// TIA Portal V17 export
// export: Created 2023-05-12T10:40:25.6107869Z, DisplayName Totally Integrated Automation Portal, DisplayVersion V17 Update 4, DisplayName TIA Portal Openness, DisplayVersion V17 Update 4, DisplayName TIA Portal Version Control Interface, DisplayVersion V17, DisplayName STEP 7 Professional, DisplayVersion V17 Update 4, DisplayName STEP 7 Safety, DisplayVersion V17, DisplayName WinCC Advanced / Unified PC, DisplayVersion V17 Update 4
FUNCTION_BLOCK "FB_EM_InputConditioning"   // FB19, LAD
{ S7_Optimized_Access := 'TRUE' }
VERSION : 0.1
// stored: AutoNumber true, CodeModifiedDate 2023-05-12T12:59:41.6492354Z, CompileDate 2023-05-12T12:59:41.6492354Z, CreationDate 2023-05-08T12:19:11.3376827Z, DownloadWithoutReinit false, HandleErrorsWithinBlock false, InterfaceModifiedDate 2023-05-12T12:59:19.7337351Z, IsConsistent true, IsIECCheckEnabled false, IsKnowHowProtected false, IsRetainMemResEnabled false, IsWriteProtected false, LibraryConformanceStatus Warning: The object contains access to global data blocks., MemoryReserve 100, ModifiedDate 2023-05-12T12:59:41.6492354Z, ParameterModified 2022-09-13T10:25:33.4387708Z, PLCSimAdvancedSupport true, SetENOAutomatically false, StructureModified 2023-05-12T12:59:19.7337351Z, UDAEnableTagReadback false
   VAR
      TT01_TempZasil_PLD3_Inst { S7_SetPoint := 'True'} : "FB_CM_MeasurementPoint";
      TT02_TempPowr_PLD3_Inst { S7_SetPoint := 'True'} : "FB_CM_MeasurementPoint";
      PT01_CisnZasil_PLD3_Inst { S7_SetPoint := 'True'} : "FB_CM_MeasurementPoint";
      PT02_CisnPowr_PLD3_Inst { S7_SetPoint := 'True'} : "FB_CM_MeasurementPoint";
      PT03_CisnZasil_JKK20_Inst { S7_SetPoint := 'True'} : "FB_CM_MeasurementPoint";
      PT04_CisnPowr_JKK20_Inst { S7_SetPoint := 'True'} : "FB_CM_MeasurementPoint";
      TTs_TempSzafy_Inst { S7_SetPoint := 'True'} : "FB_CM_MeasurementPoint";
      TTk_TempKom_Inst { S7_SetPoint := 'True'} : "FB_CM_MeasurementPoint";
      TTz_TempZewn_Inst { S7_SetPoint := 'True'} : "FB_CM_MeasurementPoint";
      Rezerwa1_Inst { S7_SetPoint := 'True'} : "FB_CM_MeasurementPoint";
      Rezerwa2_Inst { S7_SetPoint := 'True'} : "FB_CM_MeasurementPoint";
      Rezerwa3_Inst { S7_SetPoint := 'True'} : "FB_CM_MeasurementPoint";
   END_VAR
BEGIN

REGION Network 1: TT01_TempZasil_PLD3 - Temperatura zasilania z PLD3
   // TT01_TempZasil_PLD3 - Temperatura zasilania z PLD3
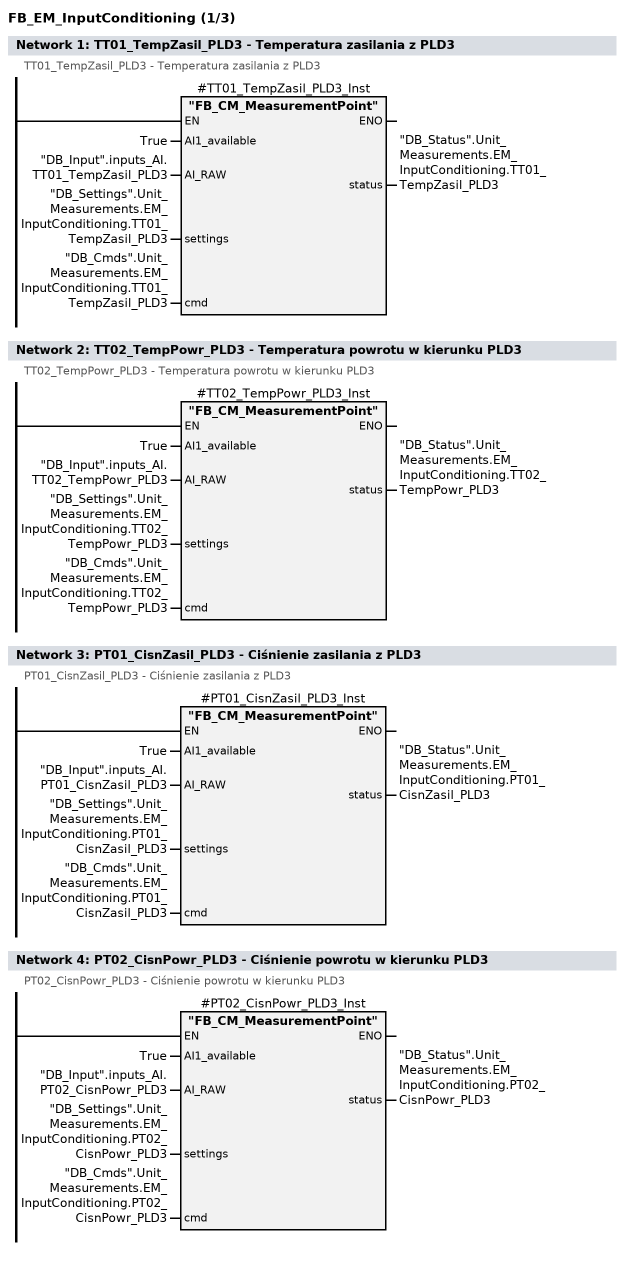
   RUNG wire#powerrail
      #TT01_TempZasil_PLD3_Inst(AI1_available := True, AI_RAW := "DB_Input".inputs_AI.TT01_TempZasil_PLD3, settings := "DB_Settings".Unit_Measurements.EM_InputConditioning.TT01_TempZasil_PLD3, cmd := "DB_Cmds".Unit_Measurements.EM_InputConditioning.TT01_TempZasil_PLD3, status => "DB_Status".Unit_Measurements.EM_InputConditioning.TT01_TempZasil_PLD3)
   END_RUNG
   // the same network as SCL:
   #TT01_TempZasil_PLD3_Inst(AI1_available := True,   // "FB_CM_MeasurementPoint"
                           AI_RAW := "DB_Input".inputs_AI.TT01_TempZasil_PLD3,
                           settings := "DB_Settings".Unit_Measurements.EM_InputConditioning.TT01_TempZasil_PLD3,
                           cmd := "DB_Cmds".Unit_Measurements.EM_InputConditioning.TT01_TempZasil_PLD3,
                           status => "DB_Status".Unit_Measurements.EM_InputConditioning.TT01_TempZasil_PLD3);
END_REGION

REGION Network 2: TT02_TempPowr_PLD3 - Temperatura powrotu w kierunku PLD3
   // TT02_TempPowr_PLD3 - Temperatura powrotu w kierunku PLD3
   RUNG wire#powerrail
      #TT02_TempPowr_PLD3_Inst(AI1_available := True, AI_RAW := "DB_Input".inputs_AI.TT02_TempPowr_PLD3, settings := "DB_Settings".Unit_Measurements.EM_InputConditioning.TT02_TempPowr_PLD3, cmd := "DB_Cmds".Unit_Measurements.EM_InputConditioning.TT02_TempPowr_PLD3, status => "DB_Status".Unit_Measurements.EM_InputConditioning.TT02_TempPowr_PLD3)
   END_RUNG
   // the same network as SCL:
   #TT02_TempPowr_PLD3_Inst(AI1_available := True,   // "FB_CM_MeasurementPoint"
                           AI_RAW := "DB_Input".inputs_AI.TT02_TempPowr_PLD3,
                           settings := "DB_Settings".Unit_Measurements.EM_InputConditioning.TT02_TempPowr_PLD3,
                           cmd := "DB_Cmds".Unit_Measurements.EM_InputConditioning.TT02_TempPowr_PLD3,
                           status => "DB_Status".Unit_Measurements.EM_InputConditioning.TT02_TempPowr_PLD3);
END_REGION

REGION Network 3: PT01_CisnZasil_PLD3 - Ciśnienie zasilania z PLD3
   // PT01_CisnZasil_PLD3 - Ciśnienie zasilania z PLD3
   RUNG wire#powerrail
      #PT01_CisnZasil_PLD3_Inst(AI1_available := True, AI_RAW := "DB_Input".inputs_AI.PT01_CisnZasil_PLD3, settings := "DB_Settings".Unit_Measurements.EM_InputConditioning.PT01_CisnZasil_PLD3, cmd := "DB_Cmds".Unit_Measurements.EM_InputConditioning.PT01_CisnZasil_PLD3, status => "DB_Status".Unit_Measurements.EM_InputConditioning.PT01_CisnZasil_PLD3)
   END_RUNG
   // the same network as SCL:
   #PT01_CisnZasil_PLD3_Inst(AI1_available := True,   // "FB_CM_MeasurementPoint"
                           AI_RAW := "DB_Input".inputs_AI.PT01_CisnZasil_PLD3,
                           settings := "DB_Settings".Unit_Measurements.EM_InputConditioning.PT01_CisnZasil_PLD3,
                           cmd := "DB_Cmds".Unit_Measurements.EM_InputConditioning.PT01_CisnZasil_PLD3,
                           status => "DB_Status".Unit_Measurements.EM_InputConditioning.PT01_CisnZasil_PLD3);
END_REGION

REGION Network 4: PT02_CisnPowr_PLD3 - Ciśnienie powrotu w kierunku PLD3
   // PT02_CisnPowr_PLD3 - Ciśnienie powrotu w kierunku PLD3
   RUNG wire#powerrail
      #PT02_CisnPowr_PLD3_Inst(AI1_available := True, AI_RAW := "DB_Input".inputs_AI.PT02_CisnPowr_PLD3, settings := "DB_Settings".Unit_Measurements.EM_InputConditioning.PT02_CisnPowr_PLD3, cmd := "DB_Cmds".Unit_Measurements.EM_InputConditioning.PT02_CisnPowr_PLD3, status => "DB_Status".Unit_Measurements.EM_InputConditioning.PT02_CisnPowr_PLD3)
   END_RUNG
   // the same network as SCL:
   #PT02_CisnPowr_PLD3_Inst(AI1_available := True,   // "FB_CM_MeasurementPoint"
                           AI_RAW := "DB_Input".inputs_AI.PT02_CisnPowr_PLD3,
                           settings := "DB_Settings".Unit_Measurements.EM_InputConditioning.PT02_CisnPowr_PLD3,
                           cmd := "DB_Cmds".Unit_Measurements.EM_InputConditioning.PT02_CisnPowr_PLD3,
                           status => "DB_Status".Unit_Measurements.EM_InputConditioning.PT02_CisnPowr_PLD3);
END_REGION

REGION Network 5: PT03_CisnZasil_JKK20 - Ciśnienie zasilania w kierunku JKK20
   // PT03_CisnZasil_JKK20 - Ciśnienie zasilania w kierunku JKK20
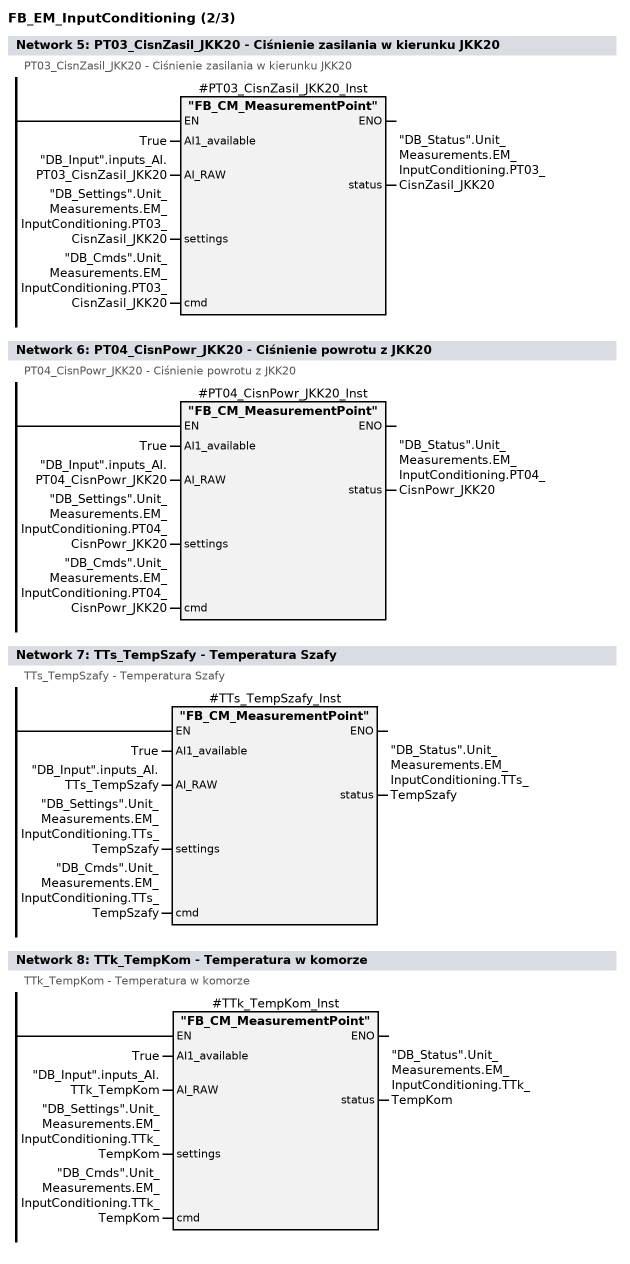
   RUNG wire#powerrail
      #PT03_CisnZasil_JKK20_Inst(AI1_available := True, AI_RAW := "DB_Input".inputs_AI.PT03_CisnZasil_JKK20, settings := "DB_Settings".Unit_Measurements.EM_InputConditioning.PT03_CisnZasil_JKK20, cmd := "DB_Cmds".Unit_Measurements.EM_InputConditioning.PT03_CisnZasil_JKK20, status => "DB_Status".Unit_Measurements.EM_InputConditioning.PT03_CisnZasil_JKK20)
   END_RUNG
   // the same network as SCL:
   #PT03_CisnZasil_JKK20_Inst(AI1_available := True,   // "FB_CM_MeasurementPoint"
                           AI_RAW := "DB_Input".inputs_AI.PT03_CisnZasil_JKK20,
                           settings := "DB_Settings".Unit_Measurements.EM_InputConditioning.PT03_CisnZasil_JKK20,
                           cmd := "DB_Cmds".Unit_Measurements.EM_InputConditioning.PT03_CisnZasil_JKK20,
                           status => "DB_Status".Unit_Measurements.EM_InputConditioning.PT03_CisnZasil_JKK20);
END_REGION

REGION Network 6: PT04_CisnPowr_JKK20 - Ciśnienie powrotu z JKK20
   // PT04_CisnPowr_JKK20 - Ciśnienie powrotu z JKK20
   RUNG wire#powerrail
      #PT04_CisnPowr_JKK20_Inst(AI1_available := True, AI_RAW := "DB_Input".inputs_AI.PT04_CisnPowr_JKK20, settings := "DB_Settings".Unit_Measurements.EM_InputConditioning.PT04_CisnPowr_JKK20, cmd := "DB_Cmds".Unit_Measurements.EM_InputConditioning.PT04_CisnPowr_JKK20, status => "DB_Status".Unit_Measurements.EM_InputConditioning.PT04_CisnPowr_JKK20)
   END_RUNG
   // the same network as SCL:
   #PT04_CisnPowr_JKK20_Inst(AI1_available := True,   // "FB_CM_MeasurementPoint"
                           AI_RAW := "DB_Input".inputs_AI.PT04_CisnPowr_JKK20,
                           settings := "DB_Settings".Unit_Measurements.EM_InputConditioning.PT04_CisnPowr_JKK20,
                           cmd := "DB_Cmds".Unit_Measurements.EM_InputConditioning.PT04_CisnPowr_JKK20,
                           status => "DB_Status".Unit_Measurements.EM_InputConditioning.PT04_CisnPowr_JKK20);
END_REGION

REGION Network 7: TTs_TempSzafy - Temperatura Szafy
   // TTs_TempSzafy - Temperatura Szafy
   RUNG wire#powerrail
      #TTs_TempSzafy_Inst(AI1_available := True, AI_RAW := "DB_Input".inputs_AI.TTs_TempSzafy, settings := "DB_Settings".Unit_Measurements.EM_InputConditioning.TTs_TempSzafy, cmd := "DB_Cmds".Unit_Measurements.EM_InputConditioning.TTs_TempSzafy, status => "DB_Status".Unit_Measurements.EM_InputConditioning.TTs_TempSzafy)
   END_RUNG
   // the same network as SCL:
   #TTs_TempSzafy_Inst(AI1_available := True,   // "FB_CM_MeasurementPoint"
                       AI_RAW := "DB_Input".inputs_AI.TTs_TempSzafy,
                       settings := "DB_Settings".Unit_Measurements.EM_InputConditioning.TTs_TempSzafy,
                       cmd := "DB_Cmds".Unit_Measurements.EM_InputConditioning.TTs_TempSzafy,
                       status => "DB_Status".Unit_Measurements.EM_InputConditioning.TTs_TempSzafy);
END_REGION

REGION Network 8: TTk_TempKom - Temperatura w komorze
   // TTk_TempKom - Temperatura w komorze
   RUNG wire#powerrail
      #TTk_TempKom_Inst(AI1_available := True, AI_RAW := "DB_Input".inputs_AI.TTk_TempKom, settings := "DB_Settings".Unit_Measurements.EM_InputConditioning.TTk_TempKom, cmd := "DB_Cmds".Unit_Measurements.EM_InputConditioning.TTk_TempKom, status => "DB_Status".Unit_Measurements.EM_InputConditioning.TTk_TempKom)
   END_RUNG
   // the same network as SCL:
   #TTk_TempKom_Inst(AI1_available := True,   // "FB_CM_MeasurementPoint"
                     AI_RAW := "DB_Input".inputs_AI.TTk_TempKom,
                     settings := "DB_Settings".Unit_Measurements.EM_InputConditioning.TTk_TempKom,
                     cmd := "DB_Cmds".Unit_Measurements.EM_InputConditioning.TTk_TempKom,
                     status => "DB_Status".Unit_Measurements.EM_InputConditioning.TTk_TempKom);
END_REGION

REGION Network 9: TTz_TempZewn - Temperatura zewnętrzna
   // TTz_TempZewn - Temperatura zewnętrzna
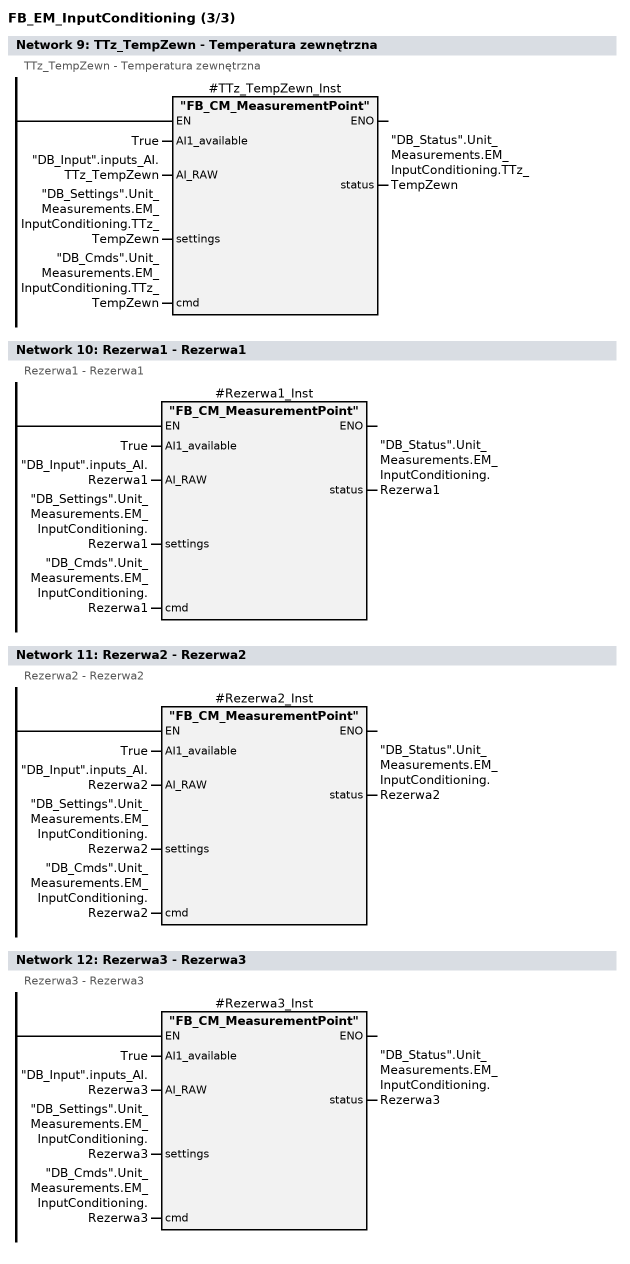
   RUNG wire#powerrail
      #TTz_TempZewn_Inst(AI1_available := True, AI_RAW := "DB_Input".inputs_AI.TTz_TempZewn, settings := "DB_Settings".Unit_Measurements.EM_InputConditioning.TTz_TempZewn, cmd := "DB_Cmds".Unit_Measurements.EM_InputConditioning.TTz_TempZewn, status => "DB_Status".Unit_Measurements.EM_InputConditioning.TTz_TempZewn)
   END_RUNG
   // the same network as SCL:
   #TTz_TempZewn_Inst(AI1_available := True,   // "FB_CM_MeasurementPoint"
                      AI_RAW := "DB_Input".inputs_AI.TTz_TempZewn,
                      settings := "DB_Settings".Unit_Measurements.EM_InputConditioning.TTz_TempZewn,
                      cmd := "DB_Cmds".Unit_Measurements.EM_InputConditioning.TTz_TempZewn,
                      status => "DB_Status".Unit_Measurements.EM_InputConditioning.TTz_TempZewn);
END_REGION

REGION Network 10: Rezerwa1 - Rezerwa1
   // Rezerwa1 - Rezerwa1
   RUNG wire#powerrail
      #Rezerwa1_Inst(AI1_available := True, AI_RAW := "DB_Input".inputs_AI.Rezerwa1, settings := "DB_Settings".Unit_Measurements.EM_InputConditioning.Rezerwa1, cmd := "DB_Cmds".Unit_Measurements.EM_InputConditioning.Rezerwa1, status => "DB_Status".Unit_Measurements.EM_InputConditioning.Rezerwa1)
   END_RUNG
   // the same network as SCL:
   #Rezerwa1_Inst(AI1_available := True,   // "FB_CM_MeasurementPoint"
                  AI_RAW := "DB_Input".inputs_AI.Rezerwa1,
                  settings := "DB_Settings".Unit_Measurements.EM_InputConditioning.Rezerwa1,
                  cmd := "DB_Cmds".Unit_Measurements.EM_InputConditioning.Rezerwa1,
                  status => "DB_Status".Unit_Measurements.EM_InputConditioning.Rezerwa1);
END_REGION

REGION Network 11: Rezerwa2 - Rezerwa2
   // Rezerwa2 - Rezerwa2
   RUNG wire#powerrail
      #Rezerwa2_Inst(AI1_available := True, AI_RAW := "DB_Input".inputs_AI.Rezerwa2, settings := "DB_Settings".Unit_Measurements.EM_InputConditioning.Rezerwa2, cmd := "DB_Cmds".Unit_Measurements.EM_InputConditioning.Rezerwa2, status => "DB_Status".Unit_Measurements.EM_InputConditioning.Rezerwa2)
   END_RUNG
   // the same network as SCL:
   #Rezerwa2_Inst(AI1_available := True,   // "FB_CM_MeasurementPoint"
                  AI_RAW := "DB_Input".inputs_AI.Rezerwa2,
                  settings := "DB_Settings".Unit_Measurements.EM_InputConditioning.Rezerwa2,
                  cmd := "DB_Cmds".Unit_Measurements.EM_InputConditioning.Rezerwa2,
                  status => "DB_Status".Unit_Measurements.EM_InputConditioning.Rezerwa2);
END_REGION

REGION Network 12: Rezerwa3 - Rezerwa3
   // Rezerwa3 - Rezerwa3
   RUNG wire#powerrail
      #Rezerwa3_Inst(AI1_available := True, AI_RAW := "DB_Input".inputs_AI.Rezerwa3, settings := "DB_Settings".Unit_Measurements.EM_InputConditioning.Rezerwa3, cmd := "DB_Cmds".Unit_Measurements.EM_InputConditioning.Rezerwa3, status => "DB_Status".Unit_Measurements.EM_InputConditioning.Rezerwa3)
   END_RUNG
   // the same network as SCL:
   #Rezerwa3_Inst(AI1_available := True,   // "FB_CM_MeasurementPoint"
                  AI_RAW := "DB_Input".inputs_AI.Rezerwa3,
                  settings := "DB_Settings".Unit_Measurements.EM_InputConditioning.Rezerwa3,
                  cmd := "DB_Cmds".Unit_Measurements.EM_InputConditioning.Rezerwa3,
                  status => "DB_Status".Unit_Measurements.EM_InputConditioning.Rezerwa3);
END_REGION
END_FUNCTION_BLOCK
